SUBAPPLICATION Uebung_102 (* DigitalInput_I1 auf DigitalOutput_Q1, mit Plug and Socket *)
  (* Standard: 61499-2 *)
  (* Version 1.0, 2023-10-23, franz *)
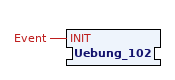
  EVENT_INPUT
    INIT;
  END_EVENT
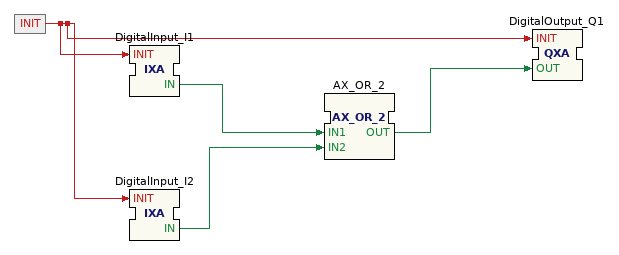
  FBS
    DigitalInput_I1 : IXA;
    DigitalOutput_Q1 : QXA;
    AX_OR_2 : io::adp::boolean::AX_OR_2;
    DigitalInput_I2 : IXA;
  END_FBS
  EVENT_CONNECTIONS
    INIT TO DigitalInput_I1.INIT;
    INIT TO DigitalOutput_Q1.INIT;
    INIT TO DigitalInput_I2.INIT;
  END_CONNECTIONS
  ADAPTER_CONNECTIONS
    AX_OR_2.OUT TO DigitalOutput_Q1.OUT;
    DigitalInput_I1.IN TO AX_OR_2.IN1;
    DigitalInput_I2.IN TO AX_OR_2.IN2;
  END_CONNECTIONS
END_SUBAPPLICATION
